// TIA Portal V17 export
// export: Created 2023-02-14T02:49:22.690637Z, ExportSetting WithDefaults, DisplayName Totally Integrated Automation Portal, DisplayVersion V17, DisplayName TIA Portal Openness, DisplayVersion V17, DisplayName TIA Portal Teamcenter Gateway, DisplayVersion V17, DisplayName TIA Portal Version Control Interface, DisplayVersion V17, DisplayName SINAMICS Startdrive Advanced, DisplayVersion V17, DisplayName SINAMICS Startdrive G130, G150, S120, S150, SINAMICS MV, S210, DisplayVersion V17, DisplayName SINAMICS Startdrive G110M, G120, G120C, G120D, G120P, G115D, DisplayVersion V17, DisplayName STEP 7 Professional, DisplayVersion V17, DisplayName STEP 7 Safety, DisplayVersion V17, DisplayName WinCC Professional, DisplayVersion V17
FUNCTION_BLOCK "IO Valve Homomixer"   // FB3, LAD
{ S7_Optimized_Access := 'FALSE' }
VERSION : 0.1
// stored: AutoNumber true, IsIECCheckEnabled false, SetENOAutomatically false, UDAEnableTagReadback false
   VAR_INPUT
      lock : Bool;
      Init : Bool;
      testing : Bool;
      Reset : Bool;
   END_VAR
   VAR
      "AV-12.01" { S7_SetPoint := 'True'} : "Valve";
      "AV-12.02" { S7_SetPoint := 'True'} : "Valve";
      "AV-12.03" { S7_SetPoint := 'True'} : "Valve";
      "AV-12.04" { S7_SetPoint := 'True'} : "Valve";
      "AV-12.05" { S7_SetPoint := 'True'} : "Valve";
      "AV-12.06" { S7_SetPoint := 'True'} : "Valve";
      "AV-12.07" { S7_SetPoint := 'True'} : "Valve";
      "AV-12.11" { S7_SetPoint := 'True'} : "Valve";
      "AV-12.12" { S7_SetPoint := 'True'} : "Valve";
      "AV-13.01" { S7_SetPoint := 'True'} : "Valve";
      "AV-13.02" { S7_SetPoint := 'True'} : "Valve";
      "AV-13.03" { S7_SetPoint := 'True'} : "Valve";
      "AV-13.04" { S7_SetPoint := 'True'} : "Valve";
      "AV-13.05" { S7_SetPoint := 'True'} : "Valve";
      "AV-13.06" { S7_SetPoint := 'True'} : "Valve";
      "AV-13.07" { S7_SetPoint := 'True'} : "Valve";
      "AV-14.01" { S7_SetPoint := 'True'} : "Valve";
      "AV-14.02" { S7_SetPoint := 'True'} : "Valve";
      "AV-14.03" { S7_SetPoint := 'True'} : "Valve";
      "AV-14.04" { S7_SetPoint := 'True'} : "Valve";
      "AV-14.05" { S7_SetPoint := 'True'} : "Valve";
      "AV-14.06" { S7_SetPoint := 'True'} : "Valve";
      "AV-14.07" { S7_SetPoint := 'True'} : "Valve";
      "P-12.01" { S7_SetPoint := 'True'} : "Motor";
      "P-13.01" { S7_SetPoint := 'True'} : "Motor";
      "P-14.01" { S7_SetPoint := 'True'} : "Motor";
   END_VAR
   // "AV-12.01".OPdwCmd := 16#0008_0000;
   // "AV-12.02".OPdwCmd := 16#0008_0000;
   // "AV-12.03".OPdwCmd := 16#0002_0000;
   // "AV-12.04".OPdwCmd := 16#0008_0000;
   // "AV-13.01".OPdwCmd := 16#0008_0000;
   // "AV-13.02".OPdwCmd := 16#0008_0000;
   // "AV-13.03".OPdwCmd := 16#0002_0000;
BEGIN

REGION Network 1 (SCL): FB OPEN and CLOSE 12
   IF #testing THEN
       // Statement section IF
       #"AV-12.01".FB_OPEN := #"AV-12.01".QCMD_OP;
       #"AV-12.01".FB_CLOSE := NOT #"AV-12.01".QCMD_OP;
       #"AV-12.02".FB_OPEN := #"AV-12.02".QCMD_OP;
       #"AV-12.02".FB_CLOSE := NOT #"AV-12.02".QCMD_OP;
       #"AV-12.03".FB_OPEN := #"AV-12.03".QCMD_OP;
       #"AV-12.03".FB_CLOSE := NOT #"AV-12.03".QCMD_OP;
       #"AV-12.04".FB_OPEN := #"AV-12.04".QCMD_OP;
       #"AV-12.04".FB_CLOSE := NOT #"AV-12.04".QCMD_OP;
       #"AV-12.05".FB_OPEN := #"AV-12.05".QCMD_OP;
       #"AV-12.05".FB_CLOSE := NOT #"AV-12.05".QCMD_OP;
       #"AV-12.06".FB_OPEN := #"AV-12.06".QCMD_OP;
       #"AV-12.06".FB_CLOSE := NOT #"AV-12.06".QCMD_OP;
       #"AV-12.07".FB_OPEN := #"AV-12.07".QCMD_OP;
       #"AV-12.07".FB_CLOSE := NOT #"AV-12.07".QCMD_OP;
       #"AV-12.11".FB_OPEN := #"AV-12.11".QCMD_OP;
       #"AV-12.11".FB_CLOSE := NOT #"AV-12.11".QCMD_OP;
       #"AV-12.12".FB_OPEN := #"AV-12.12".QCMD_OP;
       #"AV-12.12".FB_CLOSE := NOT #"AV-12.12".QCMD_OP;
   ELSE
       // Statement section ELSE
       #"AV-12.01".FB_OPEN := NOT "ZSC-12.01";
       #"AV-12.01".FB_CLOSE := "ZSC-12.01";
       #"AV-12.02".FB_OPEN := NOT "ZSC-12.02";
       #"AV-12.02".FB_CLOSE := "ZSC-12.02";
       #"AV-12.03".FB_OPEN := #"AV-12.03".QCMD_OP;
       #"AV-12.03".FB_CLOSE := NOT #"AV-12.03".QCMD_OP;
       #"AV-12.04".FB_OPEN := #"AV-12.04".QCMD_OP;
       #"AV-12.04".FB_CLOSE := NOT #"AV-12.04".QCMD_OP;
       #"AV-12.05".FB_OPEN := #"AV-12.05".QCMD_OP;
       #"AV-12.05".FB_CLOSE := NOT #"AV-12.05".QCMD_OP;
       #"AV-12.06".FB_OPEN := #"AV-12.06".QCMD_OP;
       #"AV-12.06".FB_CLOSE := NOT #"AV-12.06".QCMD_OP;
       #"AV-12.07".FB_OPEN := #"AV-12.07".QCMD_OP;
       #"AV-12.07".FB_CLOSE := NOT #"AV-12.07".QCMD_OP;
       #"AV-12.11".FB_OPEN := #"AV-12.11".QCMD_OP;
       #"AV-12.11".FB_CLOSE := NOT #"AV-12.11".QCMD_OP;
       #"AV-12.12".FB_OPEN := #"AV-12.12".QCMD_OP;
       #"AV-12.12".FB_CLOSE := NOT #"AV-12.12".QCMD_OP;
   END_IF;
END_REGION

NETWORK
TITLE = FB Monitoring Time 12
// FB OPEN Time
      L     t#20s;
      T     #"AV-12.01".MON_T;
      T     #"AV-12.02".MON_T;
      T     #"AV-12.03".MON_T;
      T     #"AV-12.04".MON_T;
      T     #"AV-12.05".MON_T;
      T     #"AV-12.06".MON_T;
      T     #"AV-12.07".MON_T;
      T     #"AV-12.11".MON_T;
      T     #"AV-12.12".MON_T;
// FB CLOSE Time
      L     t#20s;
      T     #"AV-12.01".MON_T_CLOSE;
      T     #"AV-12.02".MON_T_CLOSE;
      T     #"AV-12.03".MON_T_CLOSE;
      T     #"AV-12.04".MON_T_CLOSE;
      T     #"AV-12.05".MON_T_CLOSE;
      T     #"AV-12.06".MON_T_CLOSE;
      T     #"AV-12.07".MON_T_CLOSE;
      T     #"AV-12.11".MON_T_CLOSE;
      T     #"AV-12.12".MON_T_CLOSE;

REGION Network 3: AV-12.01 w ZSC
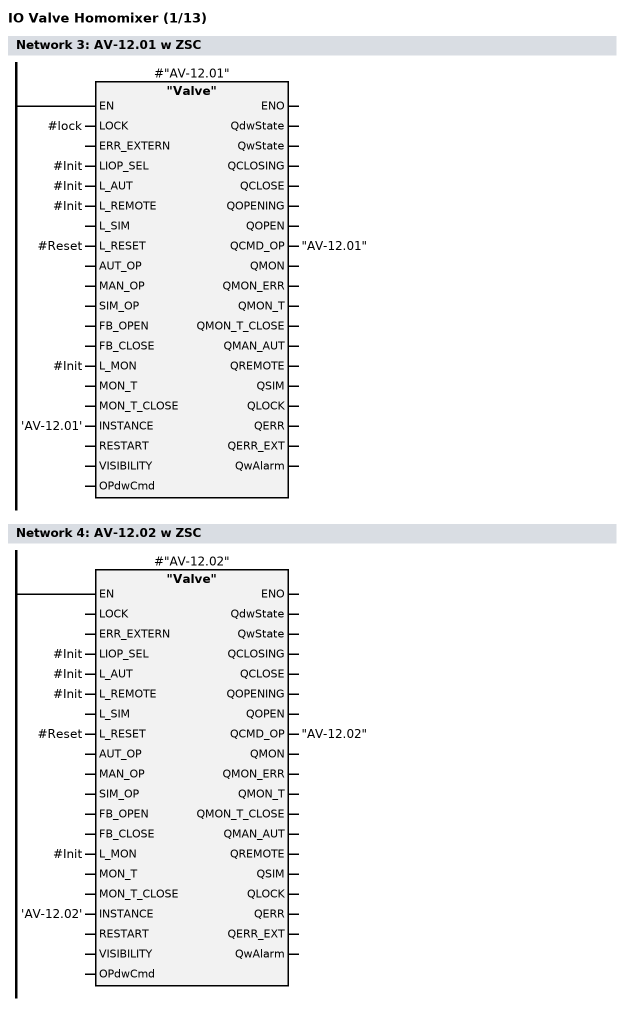
   RUNG wire#powerrail
      #"AV-12.01"(LOCK := #lock, ERR_EXTERN :=, LIOP_SEL := #Init, L_AUT := #Init, L_REMOTE := #Init, L_SIM :=, L_RESET := #Reset, AUT_OP :=, MAN_OP :=, SIM_OP :=, FB_OPEN :=, FB_CLOSE :=, L_MON := #Init, MON_T :=, MON_T_CLOSE :=, INSTANCE := 'AV-12.01', RESTART :=, VISIBILITY :=, OPdwCmd :=, QdwState =>, QwState =>, QCLOSING =>, QCLOSE =>, QOPENING =>, QOPEN =>, QCMD_OP => "AV-12.01", QMON =>, QMON_ERR =>, QMON_T =>, QMON_T_CLOSE =>, QMAN_AUT =>, QREMOTE =>, QSIM =>, QLOCK =>, QERR =>, QERR_EXT =>, QwAlarm =>)
   END_RUNG
   // the same network as SCL:
   #"AV-12.01"(LOCK := #lock,   // "Valve"
               LIOP_SEL := #Init,
               L_AUT := #Init,
               L_REMOTE := #Init,
               L_RESET := #Reset,
               L_MON := #Init,
               INSTANCE := 'AV-12.01',
               QCMD_OP => "AV-12.01");
END_REGION

REGION Network 4: AV-12.02 w ZSC
   RUNG wire#powerrail
      #"AV-12.02"(LOCK :=, ERR_EXTERN :=, LIOP_SEL := #Init, L_AUT := #Init, L_REMOTE := #Init, L_SIM :=, L_RESET := #Reset, AUT_OP :=, MAN_OP :=, SIM_OP :=, FB_OPEN :=, FB_CLOSE :=, L_MON := #Init, MON_T :=, MON_T_CLOSE :=, INSTANCE := 'AV-12.02', RESTART :=, VISIBILITY :=, OPdwCmd :=, QdwState =>, QwState =>, QCLOSING =>, QCLOSE =>, QOPENING =>, QOPEN =>, QCMD_OP => "AV-12.02", QMON =>, QMON_ERR =>, QMON_T =>, QMON_T_CLOSE =>, QMAN_AUT =>, QREMOTE =>, QSIM =>, QLOCK =>, QERR =>, QERR_EXT =>, QwAlarm =>)
   END_RUNG
   // the same network as SCL:
   #"AV-12.02"(LIOP_SEL := #Init,   // "Valve"
               L_AUT := #Init,
               L_REMOTE := #Init,
               L_RESET := #Reset,
               L_MON := #Init,
               INSTANCE := 'AV-12.02',
               QCMD_OP => "AV-12.02");
END_REGION

REGION Network 5: AV-12.03
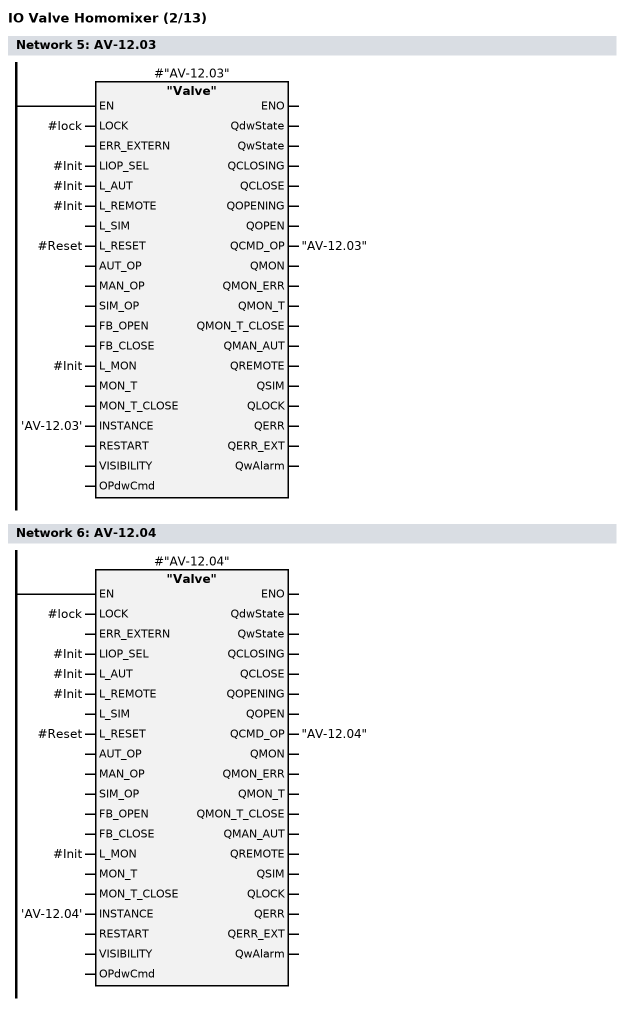
   RUNG wire#powerrail
      #"AV-12.03"(LOCK := #lock, ERR_EXTERN :=, LIOP_SEL := #Init, L_AUT := #Init, L_REMOTE := #Init, L_SIM :=, L_RESET := #Reset, AUT_OP :=, MAN_OP :=, SIM_OP :=, FB_OPEN :=, FB_CLOSE :=, L_MON := #Init, MON_T :=, MON_T_CLOSE :=, INSTANCE := 'AV-12.03', RESTART :=, VISIBILITY :=, OPdwCmd :=, QdwState =>, QwState =>, QCLOSING =>, QCLOSE =>, QOPENING =>, QOPEN =>, QCMD_OP => "AV-12.03", QMON =>, QMON_ERR =>, QMON_T =>, QMON_T_CLOSE =>, QMAN_AUT =>, QREMOTE =>, QSIM =>, QLOCK =>, QERR =>, QERR_EXT =>, QwAlarm =>)
   END_RUNG
   // the same network as SCL:
   #"AV-12.03"(LOCK := #lock,   // "Valve"
               LIOP_SEL := #Init,
               L_AUT := #Init,
               L_REMOTE := #Init,
               L_RESET := #Reset,
               L_MON := #Init,
               INSTANCE := 'AV-12.03',
               QCMD_OP => "AV-12.03");
END_REGION

REGION Network 6: AV-12.04
   RUNG wire#powerrail
      #"AV-12.04"(LOCK := #lock, ERR_EXTERN :=, LIOP_SEL := #Init, L_AUT := #Init, L_REMOTE := #Init, L_SIM :=, L_RESET := #Reset, AUT_OP :=, MAN_OP :=, SIM_OP :=, FB_OPEN :=, FB_CLOSE :=, L_MON := #Init, MON_T :=, MON_T_CLOSE :=, INSTANCE := 'AV-12.04', RESTART :=, VISIBILITY :=, OPdwCmd :=, QdwState =>, QwState =>, QCLOSING =>, QCLOSE =>, QOPENING =>, QOPEN =>, QCMD_OP => "AV-12.04", QMON =>, QMON_ERR =>, QMON_T =>, QMON_T_CLOSE =>, QMAN_AUT =>, QREMOTE =>, QSIM =>, QLOCK =>, QERR =>, QERR_EXT =>, QwAlarm =>)
   END_RUNG
   // the same network as SCL:
   #"AV-12.04"(LOCK := #lock,   // "Valve"
               LIOP_SEL := #Init,
               L_AUT := #Init,
               L_REMOTE := #Init,
               L_RESET := #Reset,
               L_MON := #Init,
               INSTANCE := 'AV-12.04',
               QCMD_OP => "AV-12.04");
END_REGION

REGION Network 7: AV-12.05
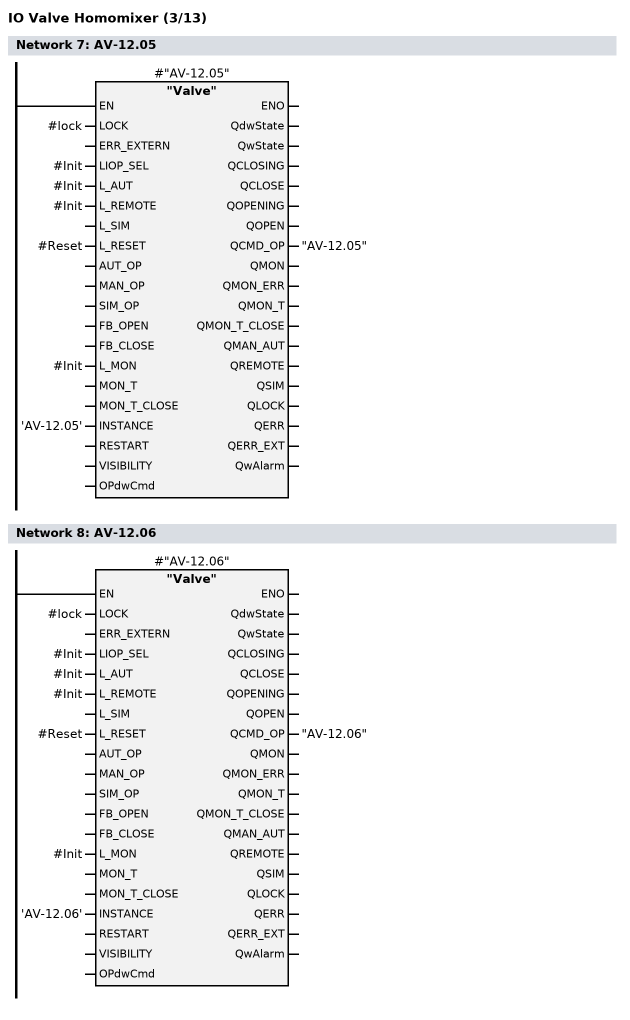
   RUNG wire#powerrail
      #"AV-12.05"(LOCK := #lock, ERR_EXTERN :=, LIOP_SEL := #Init, L_AUT := #Init, L_REMOTE := #Init, L_SIM :=, L_RESET := #Reset, AUT_OP :=, MAN_OP :=, SIM_OP :=, FB_OPEN :=, FB_CLOSE :=, L_MON := #Init, MON_T :=, MON_T_CLOSE :=, INSTANCE := 'AV-12.05', RESTART :=, VISIBILITY :=, OPdwCmd :=, QdwState =>, QwState =>, QCLOSING =>, QCLOSE =>, QOPENING =>, QOPEN =>, QCMD_OP => "AV-12.05", QMON =>, QMON_ERR =>, QMON_T =>, QMON_T_CLOSE =>, QMAN_AUT =>, QREMOTE =>, QSIM =>, QLOCK =>, QERR =>, QERR_EXT =>, QwAlarm =>)
   END_RUNG
   // the same network as SCL:
   #"AV-12.05"(LOCK := #lock,   // "Valve"
               LIOP_SEL := #Init,
               L_AUT := #Init,
               L_REMOTE := #Init,
               L_RESET := #Reset,
               L_MON := #Init,
               INSTANCE := 'AV-12.05',
               QCMD_OP => "AV-12.05");
END_REGION

REGION Network 8: AV-12.06
   RUNG wire#powerrail
      #"AV-12.06"(LOCK := #lock, ERR_EXTERN :=, LIOP_SEL := #Init, L_AUT := #Init, L_REMOTE := #Init, L_SIM :=, L_RESET := #Reset, AUT_OP :=, MAN_OP :=, SIM_OP :=, FB_OPEN :=, FB_CLOSE :=, L_MON := #Init, MON_T :=, MON_T_CLOSE :=, INSTANCE := 'AV-12.06', RESTART :=, VISIBILITY :=, OPdwCmd :=, QdwState =>, QwState =>, QCLOSING =>, QCLOSE =>, QOPENING =>, QOPEN =>, QCMD_OP => "AV-12.06", QMON =>, QMON_ERR =>, QMON_T =>, QMON_T_CLOSE =>, QMAN_AUT =>, QREMOTE =>, QSIM =>, QLOCK =>, QERR =>, QERR_EXT =>, QwAlarm =>)
   END_RUNG
   // the same network as SCL:
   #"AV-12.06"(LOCK := #lock,   // "Valve"
               LIOP_SEL := #Init,
               L_AUT := #Init,
               L_REMOTE := #Init,
               L_RESET := #Reset,
               L_MON := #Init,
               INSTANCE := 'AV-12.06',
               QCMD_OP => "AV-12.06");
END_REGION

REGION Network 9: AV-12.07
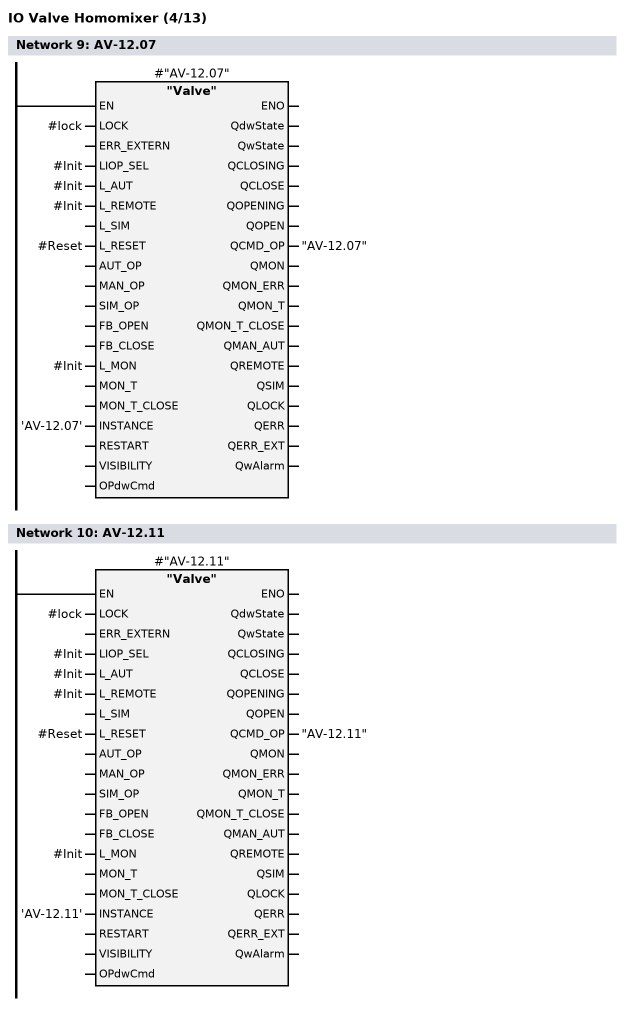
   RUNG wire#powerrail
      #"AV-12.07"(LOCK := #lock, ERR_EXTERN :=, LIOP_SEL := #Init, L_AUT := #Init, L_REMOTE := #Init, L_SIM :=, L_RESET := #Reset, AUT_OP :=, MAN_OP :=, SIM_OP :=, FB_OPEN :=, FB_CLOSE :=, L_MON := #Init, MON_T :=, MON_T_CLOSE :=, INSTANCE := 'AV-12.07', RESTART :=, VISIBILITY :=, OPdwCmd :=, QdwState =>, QwState =>, QCLOSING =>, QCLOSE =>, QOPENING =>, QOPEN =>, QCMD_OP => "AV-12.07", QMON =>, QMON_ERR =>, QMON_T =>, QMON_T_CLOSE =>, QMAN_AUT =>, QREMOTE =>, QSIM =>, QLOCK =>, QERR =>, QERR_EXT =>, QwAlarm =>)
   END_RUNG
   // the same network as SCL:
   #"AV-12.07"(LOCK := #lock,   // "Valve"
               LIOP_SEL := #Init,
               L_AUT := #Init,
               L_REMOTE := #Init,
               L_RESET := #Reset,
               L_MON := #Init,
               INSTANCE := 'AV-12.07',
               QCMD_OP => "AV-12.07");
END_REGION

REGION Network 10: AV-12.11
   RUNG wire#powerrail
      #"AV-12.11"(LOCK := #lock, ERR_EXTERN :=, LIOP_SEL := #Init, L_AUT := #Init, L_REMOTE := #Init, L_SIM :=, L_RESET := #Reset, AUT_OP :=, MAN_OP :=, SIM_OP :=, FB_OPEN :=, FB_CLOSE :=, L_MON := #Init, MON_T :=, MON_T_CLOSE :=, INSTANCE := 'AV-12.11', RESTART :=, VISIBILITY :=, OPdwCmd :=, QdwState =>, QwState =>, QCLOSING =>, QCLOSE =>, QOPENING =>, QOPEN =>, QCMD_OP => "AV-12.11", QMON =>, QMON_ERR =>, QMON_T =>, QMON_T_CLOSE =>, QMAN_AUT =>, QREMOTE =>, QSIM =>, QLOCK =>, QERR =>, QERR_EXT =>, QwAlarm =>)
   END_RUNG
   // the same network as SCL:
   #"AV-12.11"(LOCK := #lock,   // "Valve"
               LIOP_SEL := #Init,
               L_AUT := #Init,
               L_REMOTE := #Init,
               L_RESET := #Reset,
               L_MON := #Init,
               INSTANCE := 'AV-12.11',
               QCMD_OP => "AV-12.11");
END_REGION

REGION Network 11: AV-12.12
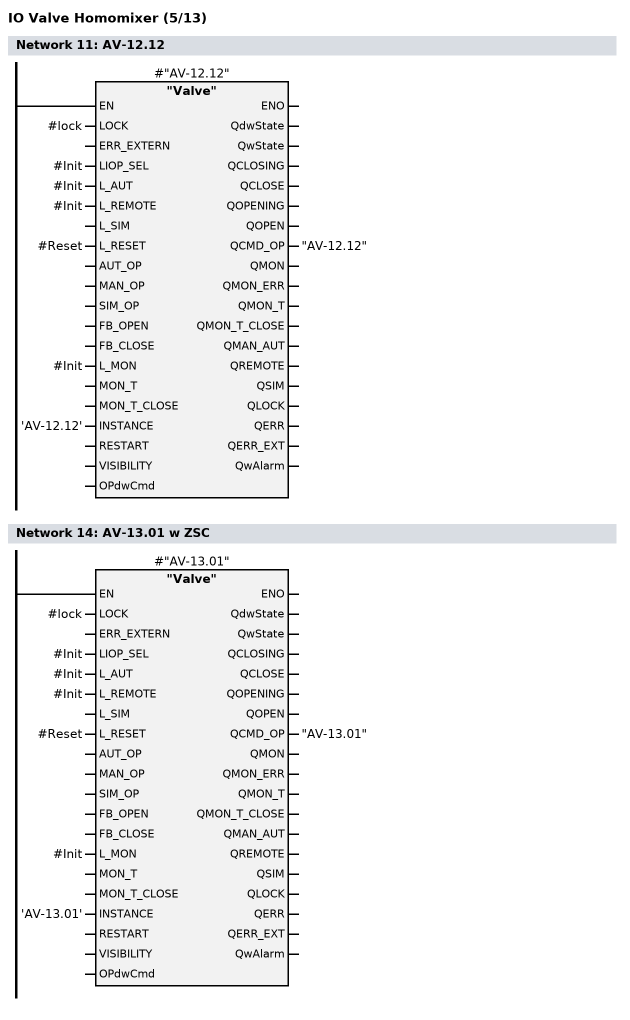
   RUNG wire#powerrail
      #"AV-12.12"(LOCK := #lock, ERR_EXTERN :=, LIOP_SEL := #Init, L_AUT := #Init, L_REMOTE := #Init, L_SIM :=, L_RESET := #Reset, AUT_OP :=, MAN_OP :=, SIM_OP :=, FB_OPEN :=, FB_CLOSE :=, L_MON := #Init, MON_T :=, MON_T_CLOSE :=, INSTANCE := 'AV-12.12', RESTART :=, VISIBILITY :=, OPdwCmd :=, QdwState =>, QwState =>, QCLOSING =>, QCLOSE =>, QOPENING =>, QOPEN =>, QCMD_OP => "AV-12.12", QMON =>, QMON_ERR =>, QMON_T =>, QMON_T_CLOSE =>, QMAN_AUT =>, QREMOTE =>, QSIM =>, QLOCK =>, QERR =>, QERR_EXT =>, QwAlarm =>)
   END_RUNG
   // the same network as SCL:
   #"AV-12.12"(LOCK := #lock,   // "Valve"
               LIOP_SEL := #Init,
               L_AUT := #Init,
               L_REMOTE := #Init,
               L_RESET := #Reset,
               L_MON := #Init,
               INSTANCE := 'AV-12.12',
               QCMD_OP => "AV-12.12");
END_REGION

REGION Network 12 (SCL): FB OPEN and CLOSE 13
   IF #testing THEN
       // Statement section IF
       #"AV-13.01".FB_OPEN := #"AV-13.01".QCMD_OP;
       #"AV-13.01".FB_CLOSE := NOT #"AV-13.01".QCMD_OP;
       #"AV-13.02".FB_OPEN := #"AV-13.02".QCMD_OP;
       #"AV-13.02".FB_CLOSE := NOT #"AV-13.02".QCMD_OP;
       #"AV-13.03".FB_OPEN := #"AV-13.03".QCMD_OP;
       #"AV-13.03".FB_CLOSE := NOT #"AV-13.03".QCMD_OP;
       #"AV-13.04".FB_OPEN := #"AV-13.04".QCMD_OP;
       #"AV-13.04".FB_CLOSE := NOT #"AV-13.04".QCMD_OP;
       #"AV-13.05".FB_OPEN := #"AV-13.05".QCMD_OP;
       #"AV-13.05".FB_CLOSE := NOT #"AV-13.05".QCMD_OP;
       #"AV-13.06".FB_OPEN := #"AV-13.06".QCMD_OP;
       #"AV-13.06".FB_CLOSE := NOT #"AV-13.06".QCMD_OP;
       #"AV-13.07".FB_OPEN := #"AV-13.07".QCMD_OP;
       #"AV-13.07".FB_CLOSE := NOT #"AV-13.07".QCMD_OP;
   ELSE
       // Statement section ELSE
       #"AV-13.01".FB_OPEN := NOT "ZSC-13.01";
       #"AV-13.01".FB_CLOSE := "ZSC-13.01";
       #"AV-13.02".FB_OPEN := NOT "ZSC-13.02";
       #"AV-13.02".FB_CLOSE := "ZSC-13.02";
       #"AV-13.03".FB_OPEN := #"AV-13.03".QCMD_OP;
       #"AV-13.03".FB_CLOSE := NOT #"AV-13.03".QCMD_OP;
       #"AV-13.04".FB_OPEN := #"AV-13.04".QCMD_OP;
       #"AV-13.04".FB_CLOSE := NOT #"AV-13.04".QCMD_OP;
       #"AV-13.05".FB_OPEN := #"AV-13.05".QCMD_OP;
       #"AV-13.05".FB_CLOSE := NOT #"AV-13.05".QCMD_OP;
       #"AV-13.06".FB_OPEN := #"AV-13.06".QCMD_OP;
       #"AV-13.06".FB_CLOSE := NOT #"AV-13.06".QCMD_OP;
       #"AV-13.07".FB_OPEN := #"AV-13.07".QCMD_OP;
       #"AV-13.07".FB_CLOSE := NOT #"AV-13.07".QCMD_OP;
   END_IF;
END_REGION

NETWORK
TITLE = FB Monitoring Time 13
// FB OPEN Time
      L     t#20s;
      T     #"AV-13.01".MON_T;
      T     #"AV-13.02".MON_T;
      T     #"AV-13.03".MON_T;
      T     #"AV-13.04".MON_T;
      T     #"AV-13.05".MON_T;
      T     #"AV-13.06".MON_T;
      T     #"AV-13.07".MON_T;
// FB CLOSE Time
      L     t#20s;
      T     #"AV-13.01".MON_T_CLOSE;
      T     #"AV-13.02".MON_T_CLOSE;
      T     #"AV-13.03".MON_T_CLOSE;
      T     #"AV-13.04".MON_T_CLOSE;
      T     #"AV-13.05".MON_T_CLOSE;
      T     #"AV-13.06".MON_T_CLOSE;
      T     #"AV-13.07".MON_T_CLOSE;

REGION Network 14: AV-13.01 w ZSC
   RUNG wire#powerrail
      #"AV-13.01"(LOCK := #lock, ERR_EXTERN :=, LIOP_SEL := #Init, L_AUT := #Init, L_REMOTE := #Init, L_SIM :=, L_RESET := #Reset, AUT_OP :=, MAN_OP :=, SIM_OP :=, FB_OPEN :=, FB_CLOSE :=, L_MON := #Init, MON_T :=, MON_T_CLOSE :=, INSTANCE := 'AV-13.01', RESTART :=, VISIBILITY :=, OPdwCmd :=, QdwState =>, QwState =>, QCLOSING =>, QCLOSE =>, QOPENING =>, QOPEN =>, QCMD_OP => "AV-13.01", QMON =>, QMON_ERR =>, QMON_T =>, QMON_T_CLOSE =>, QMAN_AUT =>, QREMOTE =>, QSIM =>, QLOCK =>, QERR =>, QERR_EXT =>, QwAlarm =>)
   END_RUNG
   // the same network as SCL:
   #"AV-13.01"(LOCK := #lock,   // "Valve"
               LIOP_SEL := #Init,
               L_AUT := #Init,
               L_REMOTE := #Init,
               L_RESET := #Reset,
               L_MON := #Init,
               INSTANCE := 'AV-13.01',
               QCMD_OP => "AV-13.01");
END_REGION

REGION Network 15: AV-13.02 w ZSC
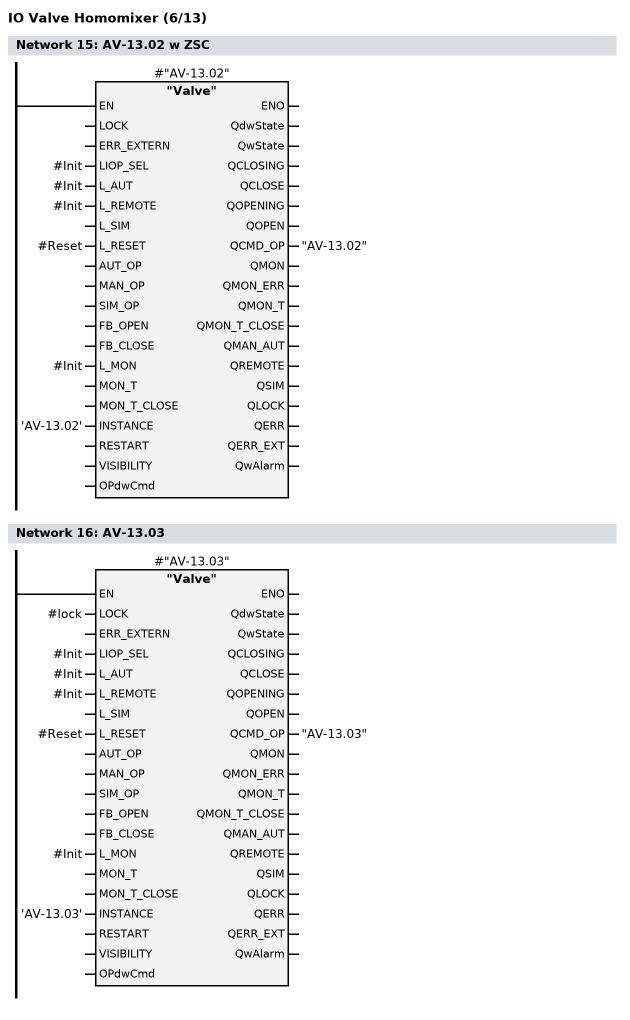
   RUNG wire#powerrail
      #"AV-13.02"(LOCK :=, ERR_EXTERN :=, LIOP_SEL := #Init, L_AUT := #Init, L_REMOTE := #Init, L_SIM :=, L_RESET := #Reset, AUT_OP :=, MAN_OP :=, SIM_OP :=, FB_OPEN :=, FB_CLOSE :=, L_MON := #Init, MON_T :=, MON_T_CLOSE :=, INSTANCE := 'AV-13.02', RESTART :=, VISIBILITY :=, OPdwCmd :=, QdwState =>, QwState =>, QCLOSING =>, QCLOSE =>, QOPENING =>, QOPEN =>, QCMD_OP => "AV-13.02", QMON =>, QMON_ERR =>, QMON_T =>, QMON_T_CLOSE =>, QMAN_AUT =>, QREMOTE =>, QSIM =>, QLOCK =>, QERR =>, QERR_EXT =>, QwAlarm =>)
   END_RUNG
   // the same network as SCL:
   #"AV-13.02"(LIOP_SEL := #Init,   // "Valve"
               L_AUT := #Init,
               L_REMOTE := #Init,
               L_RESET := #Reset,
               L_MON := #Init,
               INSTANCE := 'AV-13.02',
               QCMD_OP => "AV-13.02");
END_REGION

REGION Network 16: AV-13.03
   RUNG wire#powerrail
      #"AV-13.03"(LOCK := #lock, ERR_EXTERN :=, LIOP_SEL := #Init, L_AUT := #Init, L_REMOTE := #Init, L_SIM :=, L_RESET := #Reset, AUT_OP :=, MAN_OP :=, SIM_OP :=, FB_OPEN :=, FB_CLOSE :=, L_MON := #Init, MON_T :=, MON_T_CLOSE :=, INSTANCE := 'AV-13.03', RESTART :=, VISIBILITY :=, OPdwCmd :=, QdwState =>, QwState =>, QCLOSING =>, QCLOSE =>, QOPENING =>, QOPEN =>, QCMD_OP => "AV-13.03", QMON =>, QMON_ERR =>, QMON_T =>, QMON_T_CLOSE =>, QMAN_AUT =>, QREMOTE =>, QSIM =>, QLOCK =>, QERR =>, QERR_EXT =>, QwAlarm =>)
   END_RUNG
   // the same network as SCL:
   #"AV-13.03"(LOCK := #lock,   // "Valve"
               LIOP_SEL := #Init,
               L_AUT := #Init,
               L_REMOTE := #Init,
               L_RESET := #Reset,
               L_MON := #Init,
               INSTANCE := 'AV-13.03',
               QCMD_OP => "AV-13.03");
END_REGION

REGION Network 17: AV-13.04
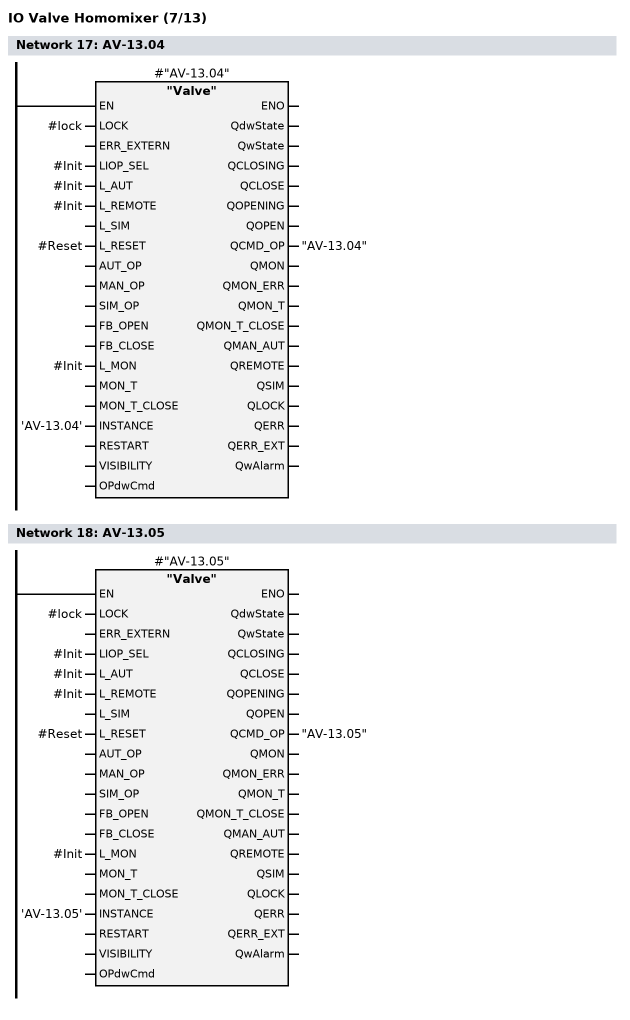
   RUNG wire#powerrail
      #"AV-13.04"(LOCK := #lock, ERR_EXTERN :=, LIOP_SEL := #Init, L_AUT := #Init, L_REMOTE := #Init, L_SIM :=, L_RESET := #Reset, AUT_OP :=, MAN_OP :=, SIM_OP :=, FB_OPEN :=, FB_CLOSE :=, L_MON := #Init, MON_T :=, MON_T_CLOSE :=, INSTANCE := 'AV-13.04', RESTART :=, VISIBILITY :=, OPdwCmd :=, QdwState =>, QwState =>, QCLOSING =>, QCLOSE =>, QOPENING =>, QOPEN =>, QCMD_OP => "AV-13.04", QMON =>, QMON_ERR =>, QMON_T =>, QMON_T_CLOSE =>, QMAN_AUT =>, QREMOTE =>, QSIM =>, QLOCK =>, QERR =>, QERR_EXT =>, QwAlarm =>)
   END_RUNG
   // the same network as SCL:
   #"AV-13.04"(LOCK := #lock,   // "Valve"
               LIOP_SEL := #Init,
               L_AUT := #Init,
               L_REMOTE := #Init,
               L_RESET := #Reset,
               L_MON := #Init,
               INSTANCE := 'AV-13.04',
               QCMD_OP => "AV-13.04");
END_REGION

REGION Network 18: AV-13.05
   RUNG wire#powerrail
      #"AV-13.05"(LOCK := #lock, ERR_EXTERN :=, LIOP_SEL := #Init, L_AUT := #Init, L_REMOTE := #Init, L_SIM :=, L_RESET := #Reset, AUT_OP :=, MAN_OP :=, SIM_OP :=, FB_OPEN :=, FB_CLOSE :=, L_MON := #Init, MON_T :=, MON_T_CLOSE :=, INSTANCE := 'AV-13.05', RESTART :=, VISIBILITY :=, OPdwCmd :=, QdwState =>, QwState =>, QCLOSING =>, QCLOSE =>, QOPENING =>, QOPEN =>, QCMD_OP => "AV-13.05", QMON =>, QMON_ERR =>, QMON_T =>, QMON_T_CLOSE =>, QMAN_AUT =>, QREMOTE =>, QSIM =>, QLOCK =>, QERR =>, QERR_EXT =>, QwAlarm =>)
   END_RUNG
   // the same network as SCL:
   #"AV-13.05"(LOCK := #lock,   // "Valve"
               LIOP_SEL := #Init,
               L_AUT := #Init,
               L_REMOTE := #Init,
               L_RESET := #Reset,
               L_MON := #Init,
               INSTANCE := 'AV-13.05',
               QCMD_OP => "AV-13.05");
END_REGION

REGION Network 19: AV-13.06
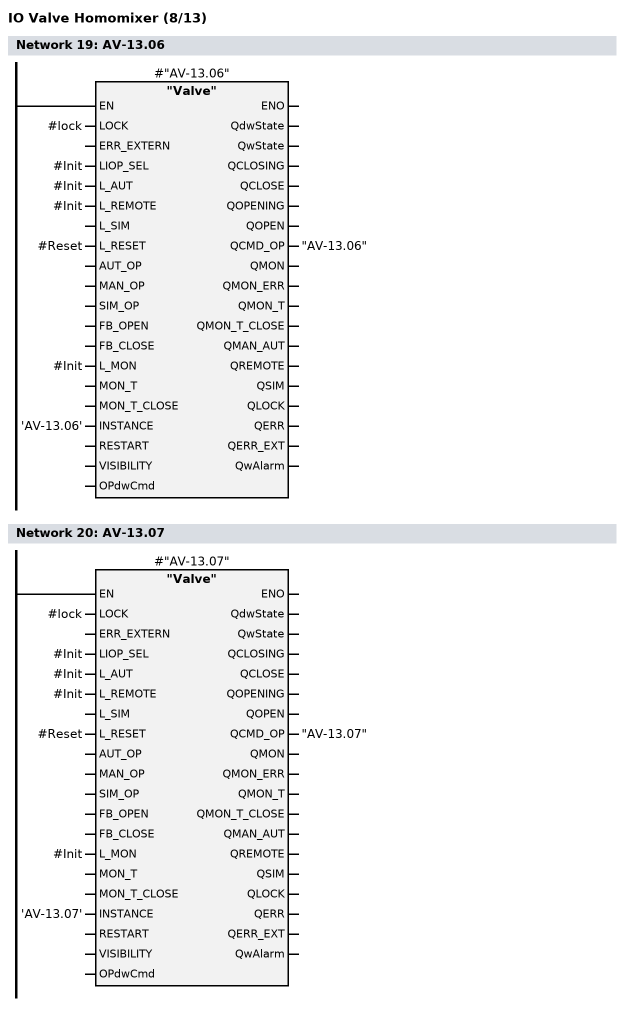
   RUNG wire#powerrail
      #"AV-13.06"(LOCK := #lock, ERR_EXTERN :=, LIOP_SEL := #Init, L_AUT := #Init, L_REMOTE := #Init, L_SIM :=, L_RESET := #Reset, AUT_OP :=, MAN_OP :=, SIM_OP :=, FB_OPEN :=, FB_CLOSE :=, L_MON := #Init, MON_T :=, MON_T_CLOSE :=, INSTANCE := 'AV-13.06', RESTART :=, VISIBILITY :=, OPdwCmd :=, QdwState =>, QwState =>, QCLOSING =>, QCLOSE =>, QOPENING =>, QOPEN =>, QCMD_OP => "AV-13.06", QMON =>, QMON_ERR =>, QMON_T =>, QMON_T_CLOSE =>, QMAN_AUT =>, QREMOTE =>, QSIM =>, QLOCK =>, QERR =>, QERR_EXT =>, QwAlarm =>)
   END_RUNG
   // the same network as SCL:
   #"AV-13.06"(LOCK := #lock,   // "Valve"
               LIOP_SEL := #Init,
               L_AUT := #Init,
               L_REMOTE := #Init,
               L_RESET := #Reset,
               L_MON := #Init,
               INSTANCE := 'AV-13.06',
               QCMD_OP => "AV-13.06");
END_REGION

REGION Network 20: AV-13.07
   RUNG wire#powerrail
      #"AV-13.07"(LOCK := #lock, ERR_EXTERN :=, LIOP_SEL := #Init, L_AUT := #Init, L_REMOTE := #Init, L_SIM :=, L_RESET := #Reset, AUT_OP :=, MAN_OP :=, SIM_OP :=, FB_OPEN :=, FB_CLOSE :=, L_MON := #Init, MON_T :=, MON_T_CLOSE :=, INSTANCE := 'AV-13.07', RESTART :=, VISIBILITY :=, OPdwCmd :=, QdwState =>, QwState =>, QCLOSING =>, QCLOSE =>, QOPENING =>, QOPEN =>, QCMD_OP => "AV-13.07", QMON =>, QMON_ERR =>, QMON_T =>, QMON_T_CLOSE =>, QMAN_AUT =>, QREMOTE =>, QSIM =>, QLOCK =>, QERR =>, QERR_EXT =>, QwAlarm =>)
   END_RUNG
   // the same network as SCL:
   #"AV-13.07"(LOCK := #lock,   // "Valve"
               LIOP_SEL := #Init,
               L_AUT := #Init,
               L_REMOTE := #Init,
               L_RESET := #Reset,
               L_MON := #Init,
               INSTANCE := 'AV-13.07',
               QCMD_OP => "AV-13.07");
END_REGION

REGION Network 21 (SCL): FB OPEN and CLOSE 14
   IF #testing THEN
       // Statement section IF
       #"AV-14.01".FB_OPEN := #"AV-14.01".QCMD_OP;
       #"AV-14.01".FB_CLOSE := NOT #"AV-14.01".QCMD_OP;
       #"AV-14.02".FB_OPEN := #"AV-14.02".QCMD_OP;
       #"AV-14.02".FB_CLOSE := NOT #"AV-14.02".QCMD_OP;
       #"AV-14.03".FB_OPEN := #"AV-14.03".QCMD_OP;
       #"AV-14.03".FB_CLOSE := NOT #"AV-14.03".QCMD_OP;
       #"AV-14.04".FB_OPEN := #"AV-14.04".QCMD_OP;
       #"AV-14.04".FB_CLOSE := NOT #"AV-14.04".QCMD_OP;
       #"AV-14.05".FB_OPEN := #"AV-14.05".QCMD_OP;
       #"AV-14.05".FB_CLOSE := NOT #"AV-14.05".QCMD_OP;
       #"AV-14.06".FB_OPEN := #"AV-14.06".QCMD_OP;
       #"AV-14.06".FB_CLOSE := NOT #"AV-14.06".QCMD_OP;
       #"AV-14.07".FB_OPEN := #"AV-14.07".QCMD_OP;
       #"AV-14.07".FB_CLOSE := NOT #"AV-14.07".QCMD_OP;
   ELSE
       // Statement section ELSE
       #"AV-14.01".FB_OPEN := NOT "ZSC-14.01";
       #"AV-14.01".FB_CLOSE := "ZSC-14.01";
       #"AV-14.02".FB_OPEN := NOT "ZSC-14.02";
       #"AV-14.02".FB_CLOSE := "ZSC-14.02";
       #"AV-14.03".FB_OPEN := #"AV-14.03".QCMD_OP;
       #"AV-14.03".FB_CLOSE := NOT #"AV-14.03".QCMD_OP;
       #"AV-14.04".FB_OPEN := #"AV-14.04".QCMD_OP;
       #"AV-14.04".FB_CLOSE := NOT #"AV-14.04".QCMD_OP;
       #"AV-14.05".FB_OPEN := #"AV-14.05".QCMD_OP;
       #"AV-14.05".FB_CLOSE := NOT #"AV-14.05".QCMD_OP;
       #"AV-14.06".FB_OPEN := #"AV-14.06".QCMD_OP;
       #"AV-14.06".FB_CLOSE := NOT #"AV-14.06".QCMD_OP;
       #"AV-14.07".FB_OPEN := #"AV-14.07".QCMD_OP;
       #"AV-14.07".FB_CLOSE := NOT #"AV-14.07".QCMD_OP;
   END_IF;
END_REGION

NETWORK
TITLE = FB Monitoring Time 14
// FB OPEN Time
      L     t#20s;
      T     #"AV-14.01".MON_T;
      T     #"AV-14.02".MON_T;
      T     #"AV-14.03".MON_T;
      T     #"AV-14.04".MON_T;
      T     #"AV-14.05".MON_T;
      T     #"AV-14.06".MON_T;
      T     #"AV-14.07".MON_T;
// FB CLOSE Time
      L     t#20s;
      T     #"AV-14.01".MON_T_CLOSE;
      T     #"AV-14.02".MON_T_CLOSE;
      T     #"AV-14.03".MON_T_CLOSE;
      T     #"AV-14.04".MON_T_CLOSE;
      T     #"AV-14.05".MON_T_CLOSE;
      T     #"AV-14.06".MON_T_CLOSE;
      T     #"AV-14.07".MON_T_CLOSE;

REGION Network 23: AV-14.01 w ZSC
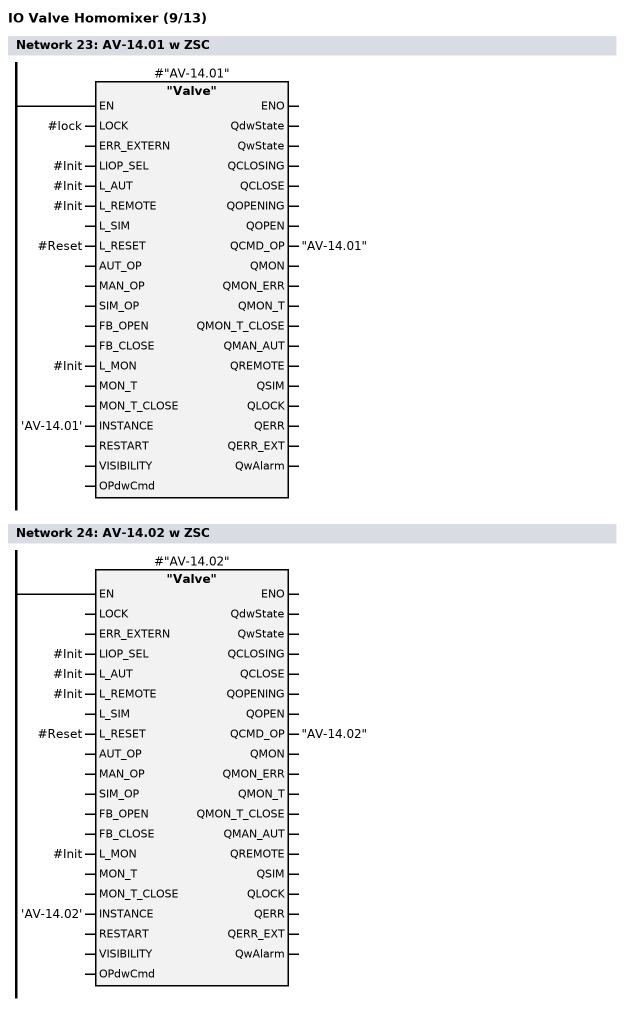
   RUNG wire#powerrail
      #"AV-14.01"(LOCK := #lock, ERR_EXTERN :=, LIOP_SEL := #Init, L_AUT := #Init, L_REMOTE := #Init, L_SIM :=, L_RESET := #Reset, AUT_OP :=, MAN_OP :=, SIM_OP :=, FB_OPEN :=, FB_CLOSE :=, L_MON := #Init, MON_T :=, MON_T_CLOSE :=, INSTANCE := 'AV-14.01', RESTART :=, VISIBILITY :=, OPdwCmd :=, QdwState =>, QwState =>, QCLOSING =>, QCLOSE =>, QOPENING =>, QOPEN =>, QCMD_OP => "AV-14.01", QMON =>, QMON_ERR =>, QMON_T =>, QMON_T_CLOSE =>, QMAN_AUT =>, QREMOTE =>, QSIM =>, QLOCK =>, QERR =>, QERR_EXT =>, QwAlarm =>)
   END_RUNG
   // the same network as SCL:
   #"AV-14.01"(LOCK := #lock,   // "Valve"
               LIOP_SEL := #Init,
               L_AUT := #Init,
               L_REMOTE := #Init,
               L_RESET := #Reset,
               L_MON := #Init,
               INSTANCE := 'AV-14.01',
               QCMD_OP => "AV-14.01");
END_REGION

REGION Network 24: AV-14.02 w ZSC
   RUNG wire#powerrail
      #"AV-14.02"(LOCK :=, ERR_EXTERN :=, LIOP_SEL := #Init, L_AUT := #Init, L_REMOTE := #Init, L_SIM :=, L_RESET := #Reset, AUT_OP :=, MAN_OP :=, SIM_OP :=, FB_OPEN :=, FB_CLOSE :=, L_MON := #Init, MON_T :=, MON_T_CLOSE :=, INSTANCE := 'AV-14.02', RESTART :=, VISIBILITY :=, OPdwCmd :=, QdwState =>, QwState =>, QCLOSING =>, QCLOSE =>, QOPENING =>, QOPEN =>, QCMD_OP => "AV-14.02", QMON =>, QMON_ERR =>, QMON_T =>, QMON_T_CLOSE =>, QMAN_AUT =>, QREMOTE =>, QSIM =>, QLOCK =>, QERR =>, QERR_EXT =>, QwAlarm =>)
   END_RUNG
   // the same network as SCL:
   #"AV-14.02"(LIOP_SEL := #Init,   // "Valve"
               L_AUT := #Init,
               L_REMOTE := #Init,
               L_RESET := #Reset,
               L_MON := #Init,
               INSTANCE := 'AV-14.02',
               QCMD_OP => "AV-14.02");
END_REGION

REGION Network 25: AV-14.03
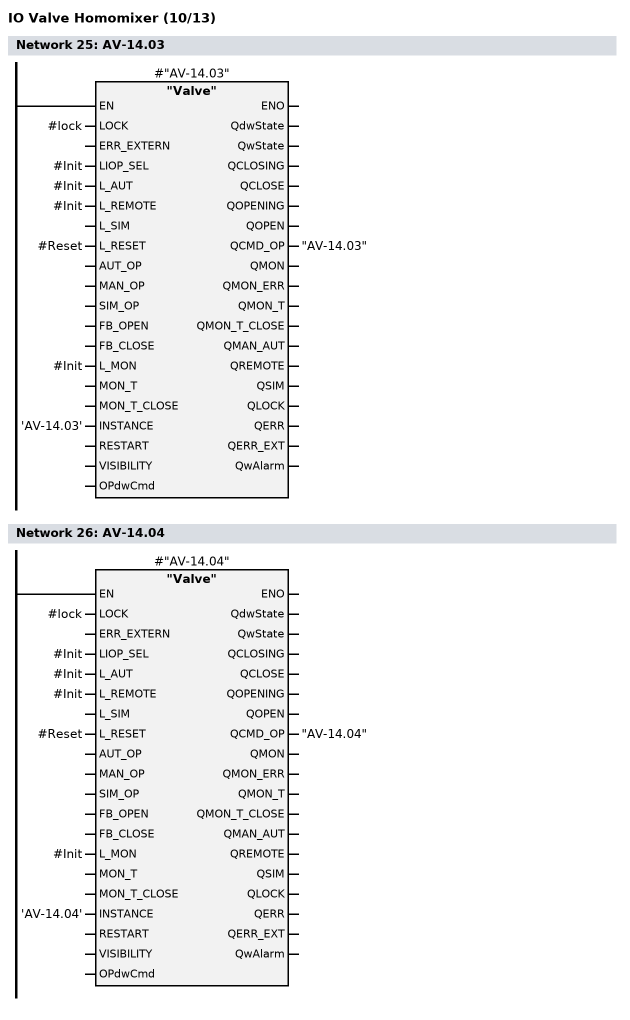
   RUNG wire#powerrail
      #"AV-14.03"(LOCK := #lock, ERR_EXTERN :=, LIOP_SEL := #Init, L_AUT := #Init, L_REMOTE := #Init, L_SIM :=, L_RESET := #Reset, AUT_OP :=, MAN_OP :=, SIM_OP :=, FB_OPEN :=, FB_CLOSE :=, L_MON := #Init, MON_T :=, MON_T_CLOSE :=, INSTANCE := 'AV-14.03', RESTART :=, VISIBILITY :=, OPdwCmd :=, QdwState =>, QwState =>, QCLOSING =>, QCLOSE =>, QOPENING =>, QOPEN =>, QCMD_OP => "AV-14.03", QMON =>, QMON_ERR =>, QMON_T =>, QMON_T_CLOSE =>, QMAN_AUT =>, QREMOTE =>, QSIM =>, QLOCK =>, QERR =>, QERR_EXT =>, QwAlarm =>)
   END_RUNG
   // the same network as SCL:
   #"AV-14.03"(LOCK := #lock,   // "Valve"
               LIOP_SEL := #Init,
               L_AUT := #Init,
               L_REMOTE := #Init,
               L_RESET := #Reset,
               L_MON := #Init,
               INSTANCE := 'AV-14.03',
               QCMD_OP => "AV-14.03");
END_REGION

REGION Network 26: AV-14.04
   RUNG wire#powerrail
      #"AV-14.04"(LOCK := #lock, ERR_EXTERN :=, LIOP_SEL := #Init, L_AUT := #Init, L_REMOTE := #Init, L_SIM :=, L_RESET := #Reset, AUT_OP :=, MAN_OP :=, SIM_OP :=, FB_OPEN :=, FB_CLOSE :=, L_MON := #Init, MON_T :=, MON_T_CLOSE :=, INSTANCE := 'AV-14.04', RESTART :=, VISIBILITY :=, OPdwCmd :=, QdwState =>, QwState =>, QCLOSING =>, QCLOSE =>, QOPENING =>, QOPEN =>, QCMD_OP => "AV-14.04", QMON =>, QMON_ERR =>, QMON_T =>, QMON_T_CLOSE =>, QMAN_AUT =>, QREMOTE =>, QSIM =>, QLOCK =>, QERR =>, QERR_EXT =>, QwAlarm =>)
   END_RUNG
   // the same network as SCL:
   #"AV-14.04"(LOCK := #lock,   // "Valve"
               LIOP_SEL := #Init,
               L_AUT := #Init,
               L_REMOTE := #Init,
               L_RESET := #Reset,
               L_MON := #Init,
               INSTANCE := 'AV-14.04',
               QCMD_OP => "AV-14.04");
END_REGION

REGION Network 27: AV-14.05
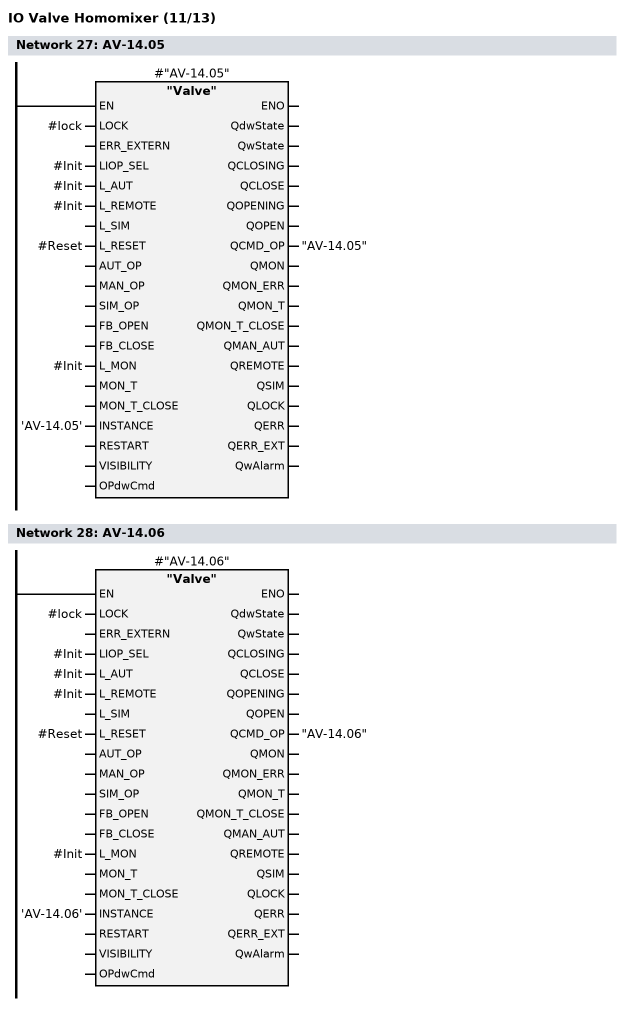
   RUNG wire#powerrail
      #"AV-14.05"(LOCK := #lock, ERR_EXTERN :=, LIOP_SEL := #Init, L_AUT := #Init, L_REMOTE := #Init, L_SIM :=, L_RESET := #Reset, AUT_OP :=, MAN_OP :=, SIM_OP :=, FB_OPEN :=, FB_CLOSE :=, L_MON := #Init, MON_T :=, MON_T_CLOSE :=, INSTANCE := 'AV-14.05', RESTART :=, VISIBILITY :=, OPdwCmd :=, QdwState =>, QwState =>, QCLOSING =>, QCLOSE =>, QOPENING =>, QOPEN =>, QCMD_OP => "AV-14.05", QMON =>, QMON_ERR =>, QMON_T =>, QMON_T_CLOSE =>, QMAN_AUT =>, QREMOTE =>, QSIM =>, QLOCK =>, QERR =>, QERR_EXT =>, QwAlarm =>)
   END_RUNG
   // the same network as SCL:
   #"AV-14.05"(LOCK := #lock,   // "Valve"
               LIOP_SEL := #Init,
               L_AUT := #Init,
               L_REMOTE := #Init,
               L_RESET := #Reset,
               L_MON := #Init,
               INSTANCE := 'AV-14.05',
               QCMD_OP => "AV-14.05");
END_REGION

REGION Network 28: AV-14.06
   RUNG wire#powerrail
      #"AV-14.06"(LOCK := #lock, ERR_EXTERN :=, LIOP_SEL := #Init, L_AUT := #Init, L_REMOTE := #Init, L_SIM :=, L_RESET := #Reset, AUT_OP :=, MAN_OP :=, SIM_OP :=, FB_OPEN :=, FB_CLOSE :=, L_MON := #Init, MON_T :=, MON_T_CLOSE :=, INSTANCE := 'AV-14.06', RESTART :=, VISIBILITY :=, OPdwCmd :=, QdwState =>, QwState =>, QCLOSING =>, QCLOSE =>, QOPENING =>, QOPEN =>, QCMD_OP => "AV-14.06", QMON =>, QMON_ERR =>, QMON_T =>, QMON_T_CLOSE =>, QMAN_AUT =>, QREMOTE =>, QSIM =>, QLOCK =>, QERR =>, QERR_EXT =>, QwAlarm =>)
   END_RUNG
   // the same network as SCL:
   #"AV-14.06"(LOCK := #lock,   // "Valve"
               LIOP_SEL := #Init,
               L_AUT := #Init,
               L_REMOTE := #Init,
               L_RESET := #Reset,
               L_MON := #Init,
               INSTANCE := 'AV-14.06',
               QCMD_OP => "AV-14.06");
END_REGION

REGION Network 29: AV-14.07
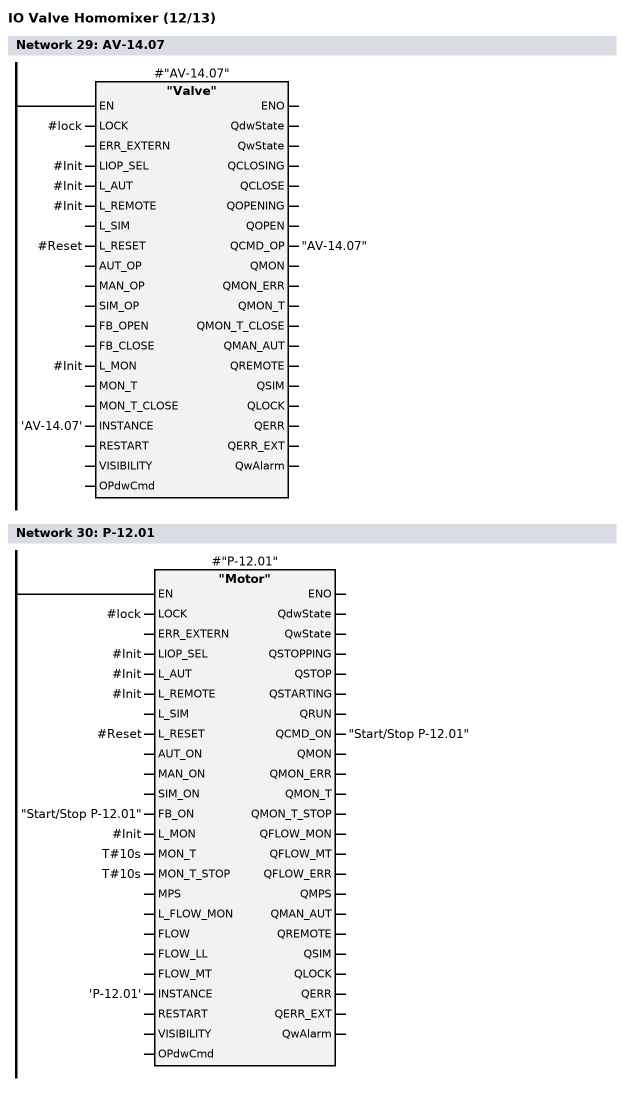
   RUNG wire#powerrail
      #"AV-14.07"(LOCK := #lock, ERR_EXTERN :=, LIOP_SEL := #Init, L_AUT := #Init, L_REMOTE := #Init, L_SIM :=, L_RESET := #Reset, AUT_OP :=, MAN_OP :=, SIM_OP :=, FB_OPEN :=, FB_CLOSE :=, L_MON := #Init, MON_T :=, MON_T_CLOSE :=, INSTANCE := 'AV-14.07', RESTART :=, VISIBILITY :=, OPdwCmd :=, QdwState =>, QwState =>, QCLOSING =>, QCLOSE =>, QOPENING =>, QOPEN =>, QCMD_OP => "AV-14.07", QMON =>, QMON_ERR =>, QMON_T =>, QMON_T_CLOSE =>, QMAN_AUT =>, QREMOTE =>, QSIM =>, QLOCK =>, QERR =>, QERR_EXT =>, QwAlarm =>)
   END_RUNG
   // the same network as SCL:
   #"AV-14.07"(LOCK := #lock,   // "Valve"
               LIOP_SEL := #Init,
               L_AUT := #Init,
               L_REMOTE := #Init,
               L_RESET := #Reset,
               L_MON := #Init,
               INSTANCE := 'AV-14.07',
               QCMD_OP => "AV-14.07");
END_REGION

REGION Network 30: P-12.01
   RUNG wire#powerrail
      #"P-12.01"(LOCK := #lock, ERR_EXTERN :=, LIOP_SEL := #Init, L_AUT := #Init, L_REMOTE := #Init, L_SIM :=, L_RESET := #Reset, AUT_ON :=, MAN_ON :=, SIM_ON :=, FB_ON := "Start/Stop P-12.01", L_MON := #Init, MON_T := T#10s, MON_T_STOP := T#10s, MPS :=, L_FLOW_MON :=, FLOW :=, FLOW_LL :=, FLOW_MT :=, INSTANCE := 'P-12.01', RESTART :=, VISIBILITY :=, OPdwCmd :=, QdwState =>, QwState =>, QSTOPPING =>, QSTOP =>, QSTARTING =>, QRUN =>, QCMD_ON => "Start/Stop P-12.01", QMON =>, QMON_ERR =>, QMON_T =>, QMON_T_STOP =>, QFLOW_MON =>, QFLOW_MT =>, QFLOW_ERR =>, QMPS =>, QMAN_AUT =>, QREMOTE =>, QSIM =>, QLOCK =>, QERR =>, QERR_EXT =>, QwAlarm =>)
   END_RUNG
   // the same network as SCL:
   #"P-12.01"(LOCK := #lock,   // "Motor"
              LIOP_SEL := #Init,
              L_AUT := #Init,
              L_REMOTE := #Init,
              L_RESET := #Reset,
              FB_ON := "Start/Stop P-12.01",
              L_MON := #Init,
              MON_T := T#10s,
              MON_T_STOP := T#10s,
              INSTANCE := 'P-12.01',
              QCMD_ON => "Start/Stop P-12.01");
END_REGION

REGION Network 31: P-13.01
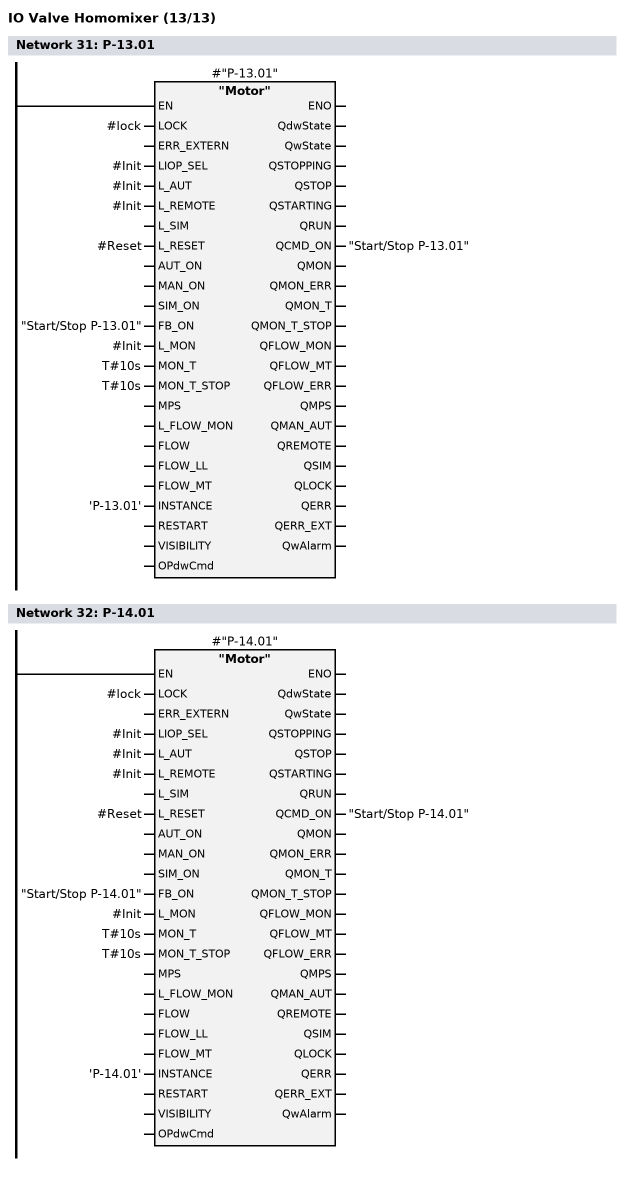
   RUNG wire#powerrail
      #"P-13.01"(LOCK := #lock, ERR_EXTERN :=, LIOP_SEL := #Init, L_AUT := #Init, L_REMOTE := #Init, L_SIM :=, L_RESET := #Reset, AUT_ON :=, MAN_ON :=, SIM_ON :=, FB_ON := "Start/Stop P-13.01", L_MON := #Init, MON_T := T#10s, MON_T_STOP := T#10s, MPS :=, L_FLOW_MON :=, FLOW :=, FLOW_LL :=, FLOW_MT :=, INSTANCE := 'P-13.01', RESTART :=, VISIBILITY :=, OPdwCmd :=, QdwState =>, QwState =>, QSTOPPING =>, QSTOP =>, QSTARTING =>, QRUN =>, QCMD_ON => "Start/Stop P-13.01", QMON =>, QMON_ERR =>, QMON_T =>, QMON_T_STOP =>, QFLOW_MON =>, QFLOW_MT =>, QFLOW_ERR =>, QMPS =>, QMAN_AUT =>, QREMOTE =>, QSIM =>, QLOCK =>, QERR =>, QERR_EXT =>, QwAlarm =>)
   END_RUNG
   // the same network as SCL:
   #"P-13.01"(LOCK := #lock,   // "Motor"
              LIOP_SEL := #Init,
              L_AUT := #Init,
              L_REMOTE := #Init,
              L_RESET := #Reset,
              FB_ON := "Start/Stop P-13.01",
              L_MON := #Init,
              MON_T := T#10s,
              MON_T_STOP := T#10s,
              INSTANCE := 'P-13.01',
              QCMD_ON => "Start/Stop P-13.01");
END_REGION

REGION Network 32: P-14.01
   RUNG wire#powerrail
      #"P-14.01"(LOCK := #lock, ERR_EXTERN :=, LIOP_SEL := #Init, L_AUT := #Init, L_REMOTE := #Init, L_SIM :=, L_RESET := #Reset, AUT_ON :=, MAN_ON :=, SIM_ON :=, FB_ON := "Start/Stop P-14.01", L_MON := #Init, MON_T := T#10s, MON_T_STOP := T#10s, MPS :=, L_FLOW_MON :=, FLOW :=, FLOW_LL :=, FLOW_MT :=, INSTANCE := 'P-14.01', RESTART :=, VISIBILITY :=, OPdwCmd :=, QdwState =>, QwState =>, QSTOPPING =>, QSTOP =>, QSTARTING =>, QRUN =>, QCMD_ON => "Start/Stop P-14.01", QMON =>, QMON_ERR =>, QMON_T =>, QMON_T_STOP =>, QFLOW_MON =>, QFLOW_MT =>, QFLOW_ERR =>, QMPS =>, QMAN_AUT =>, QREMOTE =>, QSIM =>, QLOCK =>, QERR =>, QERR_EXT =>, QwAlarm =>)
   END_RUNG
   // the same network as SCL:
   #"P-14.01"(LOCK := #lock,   // "Motor"
              LIOP_SEL := #Init,
              L_AUT := #Init,
              L_REMOTE := #Init,
              L_RESET := #Reset,
              FB_ON := "Start/Stop P-14.01",
              L_MON := #Init,
              MON_T := T#10s,
              MON_T_STOP := T#10s,
              INSTANCE := 'P-14.01',
              QCMD_ON => "Start/Stop P-14.01");
END_REGION
END_FUNCTION_BLOCK
